TYPE SafetyMotionBlockingProcesses :
STRUCT
	///Reset the errors (including the programmed ones and the TwinSAFE group ones)
	reset: Process;
END_STRUCT
END_TYPE

(* stored: Version 1.1.0.1, ProductVersion 3.1.4019.2
   DUT SafetyMotionBlockingProcesses: Id {aaa2d389-321e-4400-80c5-ea6c58d46322} *)
